Omron CX-Programmer project NewProject (CX-Programmer 9.73)

# PLC NewPLC1: CP1E N20

## Global symbols (name address type ; comment)
0.01 BOOL  ; start
0.02 BOOL  ; stop
100.00 BOOL  ; motor 1

## Program NewProgram1 (cyclic task 0)

### Section Section1

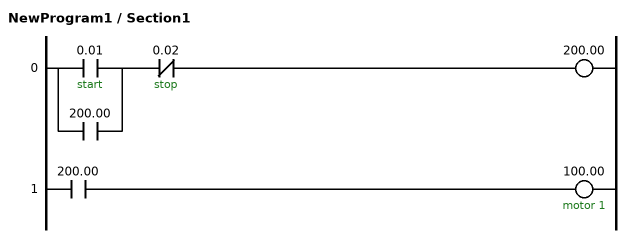
; rung 0
LD 0.01  ; start
OR 200.00
ANDNOT 0.02  ; stop
OUT 200.00
; rung 1
LD 200.00
OUT 100.00  ; motor 1

### Section END
; rung 0
END(001)